{attribute addProperty BoxType "EJ2918-0000-0017"}
{attribute addProperty Id "FSOEAT %Q*FSOE_89B9F66A567"}
{attribute addProperty CRC "1727120823"}
{attribute addProperty SizeInBites "56"}
{attribute addProperty SizeInBytes "7"}
TYPE FSoE_Outputs_66F1C5B7 :
STRUCT
	{attribute addProperty Name "FSOE"}
	FSOE AT %Q* : FSOE_89B9F66A;
END_STRUCT
END_TYPE

(* stored: Version 1.2.0.0, ProductVersion 3.1.4024.9
   DUT FSoE_Outputs_66F1C5B7: Id {3a083af5-4e69-45dd-884c-823be377e5ee} *)
